# EPICS substitutions: evgMrmApp/Db/evgSoftSeq-psi.substitutions
file evgSoftSeq.db {
pattern { P, EVG, seqNum, NELM }
{ "$(SYS):$(EVG)-SoftSeq-$(SEQNUM)-", $(EVG), 0, 2047 }
}
